{attribute 'GeneratedUsingTerminal: EK1100-0000-0018'}
{attribute addProperty BoxType "EK1100-0000-0018"}
{attribute addProperty Id "Beckhoff_EL4xxxEK1122Beckhoff_EL4xxxEK1122_243FD9A62A_0001_EL4001_0000_0016EL4001_2FC30C535A_0002_EL4001_0000_0017EL4001_2FC30C535A_0003_EL4001_0000_0018EL4001_2FC30C535A_0004_EL4001_0000_0019EL4001_2FC30C535A_0005_EL4001_0000_0020EL4001_2FC30C535A_0006_EL4002_0000_0016EL4002_CAB4C8F57A_0007_EL4002_0000_0017EL4002_CAB4C8F57A_0008_EL4002_0000_0018EL4002_D295D1387A_0009_EL4002_0000_0019EL4002_CAB4C8F57A_0010_EL4002_0000_0020EL4002_CAB4C8F57A_0011_EL4004_0000_0016EL4004_EB925BA911A_0012_EL4004_0000_0017EL4004_EB925BA911A_0013_EL4004_0000_0018EL4004_57A43C6411A_0014_EL4004_0000_0019EL4004_EB925BA911A_0015_EL4004_0000_0020EL4004_EB925BA911A_0016_EL4008_0000_0016EL4008_9E80CF7619A_0017_EL4008_0000_0017EL4008_9E80CF7619A_0018_EL4008_0000_0018EL4008_8B2492A319A_0019_EL4008_0000_0019EL4008_9E80CF7619A_0020_EL4008_0000_0020EL4008_9E80CF7619A_0021_EL4011_0000_0016EL4011_2FC30C535A_0022_EL4011_0000_0017EL4011_2FC30C535A_0023_EL4011_0000_0018EL4011_2FC30C535A_0024_EL4011_0000_0019EL4011_2FC30C535A_0025_EL4011_0000_0020EL4011_2FC30C535A_0026_EL4012_0000_0016EL4012_CAB4C8F57A_0027_EL4012_0000_0017EL4012_CAB4C8F57A_0028_EL4012_0000_0018EL4012_D295D1387A_0029_EL4012_0000_0019EL4012_CAB4C8F57A_0030_EL4012_0000_0020EL4012_CAB4C8F57A_0031_EL4014_0000_0016EL4014_EB925BA911A_0032_EL4014_0000_0017EL4014_EB925BA911A_0033_EL4014_0000_0018EL4014_57A43C6411A_0034_EL4014_0000_0019EL4014_EB925BA911A_0035_EL4014_0000_0020EL4014_EB925BA911A_0036_EL4018_0000_0016EL4018_9E80CF7619A_0037_EL4018_0000_0017EL4018_9E80CF7619A_0038_EL4018_0000_0018EL4018_8B2492A319A_0039_EL4018_0000_0019EL4018_9E80CF7619A_0040_EL4018_0000_0020EL4018_9E80CF7619A_0041_EL4021_0000_0016EL4021_2FC30C535A_0042_EL4021_0000_0017EL4021_2FC30C535A_0043_EL4021_0000_0018EL4021_2FC30C535A_0044_EL4021_0000_0019EL4021_2FC30C535A_0045_EL4021_0000_0020EL4021_2FC30C535A_0046_EL4021_0000_0021EL4021_2FC30C535A_0047_EL4022_0000_0016EL4022_CAB4C8F57A_0048_EL4022_0000_0017EL4022_CAB4C8F57A_0049_EL4022_0000_0018EL4022_D295D1387A_0050_EL4022_0000_0019EL4022_CAB4C8F57A_0051_EL4022_0000_0020EL4022_CAB4C8F57A_0052_EL4022_0000_0021EL4022_CAB4C8F57A_0053_EL4024_0000_0016EL4024_EB925BA911A_0054_EL4024_0000_0017EL4024_EB925BA911A_0055_EL4024_0000_0018EL4024_57A43C6411A_0056_EL4024_0000_0019EL4024_EB925BA911A_0057_EL4024_0000_0020EL4024_EB925BA911A_0058_EL4024_0000_0021EL4024_EB925BA911A_0059_EL4028_0000_0016EL4028_9E80CF7619A_0060_EL4028_0000_0017EL4028_9E80CF7619A_0061_EL4028_0000_0018EL4028_8B2492A319A_0062_EL4028_0000_0019EL4028_9E80CF7619A_0063_EL4028_0000_0020EL4028_9E80CF7619A_0064_EL4028_0000_0021EL4028_9E80CF7619A_0065_EL4031_0000_0016EL4031_2FC30C535A_0066_EL4031_0000_0017EL4031_2FC30C535A_0067_EL4031_0000_0018EL4031_2FC30C535A_0068_EL4031_0000_0019EL4031_2FC30C535A_0069_EL4031_0000_0020EL4031_2FC30C535A_0070_EL4032_0000_0016EL4032_CAB4C8F57A_0071_EL4032_0000_0017EL4032_CAB4C8F57A_0072_EL4032_0000_0018EL4032_D295D1387A_0073_EL4032_0000_0019EL4032_CAB4C8F57A_0074_EL4032_0000_0020EL4032_CAB4C8F57A_0075_EL4034_0000_0016EL4034_EB925BA911A_0076_EL4034_0000_0017EL4034_EB925BA911A_0077_EL4034_0000_0018EL4034_57A43C6411A_0078_EL4034_0000_0019EL4034_EB925BA911A_0079_EL4034_0000_0020EL4034_EB925BA911A_0080_EL4038_0000_0016EL4038_9E80CF7619A_0081_EL4038_0000_0017EL4038_9E80CF7619A_0082_EL4038_0000_0018EL4038_8B2492A319A_0083_EL4038_0000_0019EL4038_9E80CF7619A_0084_EL4038_0000_0020EL4038_9E80CF7619A_0085_EL4102_0000_0000EL4102_DDDE0D3B7A_0086_EL4102_0000_1016EL4102_DDDE0D3B7A_0087_EL4102_0000_1017EL4102_DDDE0D3B7A_0088_EL4102_0000_1018EL4102_DDDE0D3B7A_0089_EL4102_0000_1019EL4102_DDDE0D3B7A_0090_EL4102_0000_1020EL4102_DDDE0D3B7A_0091_EL4104_0000_1016EL4104_57A43C6411A_0092_EL4104_0000_1017EL4104_57A43C6411A_0093_EL4104_0000_1018EL4104_57A43C6411A_0094_EL4104_0000_1019EL4104_57A43C6411A_0095_EL4104_0000_1020EL4104_57A43C6411A_0096_EL4112_0000_0000EL4112_DDDE0D3B7A_0097_EL4112_0000_1016EL4112_DDDE0D3B7A_0098_EL4112_0000_1017EL4112_DDDE0D3B7A_0099_EL4112_0000_1018EL4112_DDDE0D3B7A_0100_EL4112_0000_1019EL4112_DDDE0D3B7A_0101_EL4112_0000_1020EL4112_DDDE0D3B7A_0102_EL4112_0010_0000EL4112_DDDE0D3B7A_0103_EL4112_0010_1016EL4112_DDDE0D3B7A_0104_EL4112_0010_1017EL4112_DDDE0D3B7A_0105_EL4112_0010_1018EL4112_DDDE0D3B7A_0106_EL4112_0010_1019EL4112_DDDE0D3B7A_0107_EL4112_0010_1020EL4112_DDDE0D3B7A_0108_EL4114_0000_1016EL4114_57A43C6411A_0109_EL4114_0000_1017EL4114_57A43C6411A_0110_EL4114_0000_1018EL4114_57A43C6411A_0111_EL4114_0000_1019EL4114_57A43C6411A_0112_EL4114_0000_1020EL4114_57A43C6411A_0113_EL4122_0000_0000EL4122_DDDE0D3B7A_0114_EL4122_0000_1016EL4122_DDDE0D3B7A_0115_EL4122_0000_1017EL4122_DDDE0D3B7A_0116_EL4122_0000_1018EL4122_DDDE0D3B7A_0117_EL4122_0000_1019EL4122_DDDE0D3B7A_0118_EL4122_0000_1020EL4122_DDDE0D3B7A_0119_EL4124_0000_1016EL4124_57A43C6411A_0120_EL4124_0000_1017EL4124_57A43C6411A_0121_EL4124_0000_1018EL4124_57A43C6411A_0122_EL4124_0000_1019EL4124_57A43C6411A_0123_EL4124_0000_1020EL4124_57A43C6411A_0124_EL4132_0000_0000EL4132_DDDE0D3B7A_0125_EL4132_0000_1016EL4132_DDDE0D3B7A_0126_EL4132_0000_1017EL4132_DDDE0D3B7A_0127_EL4132_0000_1018EL4132_DDDE0D3B7A_0128_EL4132_0000_1019EL4132_DDDE0D3B7A_0129_EL4132_0000_1020EL4132_DDDE0D3B7A_0130_EL4134_0000_1016EL4134_57A43C6411A_0131_EL4134_0000_1017EL4134_57A43C6411A_0132_EL4134_0000_1018EL4134_57A43C6411A_0133_EL4134_0000_1019EL4134_57A43C6411A_0134_EL4134_0000_1020EL4134_57A43C6411A_0135_EL4134_0030_1020EL4134_57A43C6411"}
{attribute addProperty CRC "2306607182"}
{attribute addProperty Size "1325"}
TYPE Beckhoff_EL4xxx_897C084E EXTENDS EK1100_1FC0878B :
STRUCT
	{attribute addProperty Name "Beckhoff_EL4xxxEK1122"}
	{attribute addProperty PreviousPort "Beckhoff EL4xxx : B"}
	Beckhoff_EL4xxxEK1122 : Beckhoff_EL4xxxEK1122_243FD9A6;
	{attribute addProperty Name "A_0001_EL4001_0000_0016"}
	{attribute addProperty PreviousPort "Beckhoff EL4xxxEK1122 : C"}
	A_0001_EL4001_0000_0016 : EL4001_2FC30C53;
	{attribute addProperty Name "A_0002_EL4001_0000_0017"}
	{attribute addProperty PreviousPort "A_0001(EL4001-0000-0016) : B"}
	A_0002_EL4001_0000_0017 : EL4001_2FC30C53;
	{attribute addProperty Name "A_0003_EL4001_0000_0018"}
	{attribute addProperty PreviousPort "A_0002(EL4001-0000-0017) : B"}
	A_0003_EL4001_0000_0018 : EL4001_2FC30C53;
	{attribute addProperty Name "A_0004_EL4001_0000_0019"}
	{attribute addProperty PreviousPort "A_0003(EL4001-0000-0018) : B"}
	A_0004_EL4001_0000_0019 : EL4001_2FC30C53;
	{attribute addProperty Name "A_0005_EL4001_0000_0020"}
	{attribute addProperty PreviousPort "A_0004(EL4001-0000-0019) : B"}
	A_0005_EL4001_0000_0020 : EL4001_2FC30C53;
	{attribute addProperty Name "A_0006_EL4002_0000_0016"}
	{attribute addProperty PreviousPort "A_0005(EL4001-0000-0020) : B"}
	A_0006_EL4002_0000_0016 : EL4002_CAB4C8F5;
	{attribute addProperty Name "A_0007_EL4002_0000_0017"}
	{attribute addProperty PreviousPort "A_0006(EL4002-0000-0016) : B"}
	A_0007_EL4002_0000_0017 : EL4002_CAB4C8F5;
	{attribute addProperty Name "A_0008_EL4002_0000_0018"}
	{attribute addProperty PreviousPort "A_0007(EL4002-0000-0017) : B"}
	A_0008_EL4002_0000_0018 : EL4002_D295D138;
	{attribute addProperty Name "A_0009_EL4002_0000_0019"}
	{attribute addProperty PreviousPort "A_0008(EL4002-0000-0018) : B"}
	A_0009_EL4002_0000_0019 : EL4002_CAB4C8F5;
	{attribute addProperty Name "A_0010_EL4002_0000_0020"}
	{attribute addProperty PreviousPort "A_0009(EL4002-0000-0019) : B"}
	A_0010_EL4002_0000_0020 : EL4002_CAB4C8F5;
	{attribute addProperty Name "A_0011_EL4004_0000_0016"}
	{attribute addProperty PreviousPort "A_0010(EL4002-0000-0020) : B"}
	A_0011_EL4004_0000_0016 : EL4004_EB925BA9;
	{attribute addProperty Name "A_0012_EL4004_0000_0017"}
	{attribute addProperty PreviousPort "A_0011(EL4004-0000-0016) : B"}
	A_0012_EL4004_0000_0017 : EL4004_EB925BA9;
	{attribute addProperty Name "A_0013_EL4004_0000_0018"}
	{attribute addProperty PreviousPort "A_0012(EL4004-0000-0017) : B"}
	A_0013_EL4004_0000_0018 : EL4004_57A43C64;
	{attribute addProperty Name "A_0014_EL4004_0000_0019"}
	{attribute addProperty PreviousPort "A_0013(EL4004-0000-0018) : B"}
	A_0014_EL4004_0000_0019 : EL4004_EB925BA9;
	{attribute addProperty Name "A_0015_EL4004_0000_0020"}
	{attribute addProperty PreviousPort "A_0014(EL4004-0000-0019) : B"}
	A_0015_EL4004_0000_0020 : EL4004_EB925BA9;
	{attribute addProperty Name "A_0016_EL4008_0000_0016"}
	{attribute addProperty PreviousPort "A_0015(EL4004-0000-0020) : B"}
	A_0016_EL4008_0000_0016 : EL4008_9E80CF76;
	{attribute addProperty Name "A_0017_EL4008_0000_0017"}
	{attribute addProperty PreviousPort "A_0016(EL4008-0000-0016) : B"}
	A_0017_EL4008_0000_0017 : EL4008_9E80CF76;
	{attribute addProperty Name "A_0018_EL4008_0000_0018"}
	{attribute addProperty PreviousPort "A_0017(EL4008-0000-0017) : B"}
	A_0018_EL4008_0000_0018 : EL4008_8B2492A3;
	{attribute addProperty Name "A_0019_EL4008_0000_0019"}
	{attribute addProperty PreviousPort "A_0018(EL4008-0000-0018) : B"}
	A_0019_EL4008_0000_0019 : EL4008_9E80CF76;
	{attribute addProperty Name "A_0020_EL4008_0000_0020"}
	{attribute addProperty PreviousPort "A_0019(EL4008-0000-0019) : B"}
	A_0020_EL4008_0000_0020 : EL4008_9E80CF76;
	{attribute addProperty Name "A_0021_EL4011_0000_0016"}
	{attribute addProperty PreviousPort "A_0020(EL4008-0000-0020) : B"}
	A_0021_EL4011_0000_0016 : EL4011_2FC30C53;
	{attribute addProperty Name "A_0022_EL4011_0000_0017"}
	{attribute addProperty PreviousPort "A_0021(EL4011-0000-0016) : B"}
	A_0022_EL4011_0000_0017 : EL4011_2FC30C53;
	{attribute addProperty Name "A_0023_EL4011_0000_0018"}
	{attribute addProperty PreviousPort "A_0022(EL4011-0000-0017) : B"}
	A_0023_EL4011_0000_0018 : EL4011_2FC30C53;
	{attribute addProperty Name "A_0024_EL4011_0000_0019"}
	{attribute addProperty PreviousPort "A_0023(EL4011-0000-0018) : B"}
	A_0024_EL4011_0000_0019 : EL4011_2FC30C53;
	{attribute addProperty Name "A_0025_EL4011_0000_0020"}
	{attribute addProperty PreviousPort "A_0024(EL4011-0000-0019) : B"}
	A_0025_EL4011_0000_0020 : EL4011_2FC30C53;
	{attribute addProperty Name "A_0026_EL4012_0000_0016"}
	{attribute addProperty PreviousPort "A_0025(EL4011-0000-0020) : B"}
	A_0026_EL4012_0000_0016 : EL4012_CAB4C8F5;
	{attribute addProperty Name "A_0027_EL4012_0000_0017"}
	{attribute addProperty PreviousPort "A_0026(EL4012-0000-0016) : B"}
	A_0027_EL4012_0000_0017 : EL4012_CAB4C8F5;
	{attribute addProperty Name "A_0028_EL4012_0000_0018"}
	{attribute addProperty PreviousPort "A_0027(EL4012-0000-0017) : B"}
	A_0028_EL4012_0000_0018 : EL4012_D295D138;
	{attribute addProperty Name "A_0029_EL4012_0000_0019"}
	{attribute addProperty PreviousPort "A_0028(EL4012-0000-0018) : B"}
	A_0029_EL4012_0000_0019 : EL4012_CAB4C8F5;
	{attribute addProperty Name "A_0030_EL4012_0000_0020"}
	{attribute addProperty PreviousPort "A_0029(EL4012-0000-0019) : B"}
	A_0030_EL4012_0000_0020 : EL4012_CAB4C8F5;
	{attribute addProperty Name "A_0031_EL4014_0000_0016"}
	{attribute addProperty PreviousPort "A_0030(EL4012-0000-0020) : B"}
	A_0031_EL4014_0000_0016 : EL4014_EB925BA9;
	{attribute addProperty Name "A_0032_EL4014_0000_0017"}
	{attribute addProperty PreviousPort "A_0031(EL4014-0000-0016) : B"}
	A_0032_EL4014_0000_0017 : EL4014_EB925BA9;
	{attribute addProperty Name "A_0033_EL4014_0000_0018"}
	{attribute addProperty PreviousPort "A_0032(EL4014-0000-0017) : B"}
	A_0033_EL4014_0000_0018 : EL4014_57A43C64;
	{attribute addProperty Name "A_0034_EL4014_0000_0019"}
	{attribute addProperty PreviousPort "A_0033(EL4014-0000-0018) : B"}
	A_0034_EL4014_0000_0019 : EL4014_EB925BA9;
	{attribute addProperty Name "A_0035_EL4014_0000_0020"}
	{attribute addProperty PreviousPort "A_0034(EL4014-0000-0019) : B"}
	A_0035_EL4014_0000_0020 : EL4014_EB925BA9;
	{attribute addProperty Name "A_0036_EL4018_0000_0016"}
	{attribute addProperty PreviousPort "A_0035(EL4014-0000-0020) : B"}
	A_0036_EL4018_0000_0016 : EL4018_9E80CF76;
	{attribute addProperty Name "A_0037_EL4018_0000_0017"}
	{attribute addProperty PreviousPort "A_0036(EL4018-0000-0016) : B"}
	A_0037_EL4018_0000_0017 : EL4018_9E80CF76;
	{attribute addProperty Name "A_0038_EL4018_0000_0018"}
	{attribute addProperty PreviousPort "A_0037(EL4018-0000-0017) : B"}
	A_0038_EL4018_0000_0018 : EL4018_8B2492A3;
	{attribute addProperty Name "A_0039_EL4018_0000_0019"}
	{attribute addProperty PreviousPort "A_0038(EL4018-0000-0018) : B"}
	A_0039_EL4018_0000_0019 : EL4018_9E80CF76;
	{attribute addProperty Name "A_0040_EL4018_0000_0020"}
	{attribute addProperty PreviousPort "A_0039(EL4018-0000-0019) : B"}
	A_0040_EL4018_0000_0020 : EL4018_9E80CF76;
	{attribute addProperty Name "A_0041_EL4021_0000_0016"}
	{attribute addProperty PreviousPort "A_0040(EL4018-0000-0020) : B"}
	A_0041_EL4021_0000_0016 : EL4021_2FC30C53;
	{attribute addProperty Name "A_0042_EL4021_0000_0017"}
	{attribute addProperty PreviousPort "A_0041(EL4021-0000-0016) : B"}
	A_0042_EL4021_0000_0017 : EL4021_2FC30C53;
	{attribute addProperty Name "A_0043_EL4021_0000_0018"}
	{attribute addProperty PreviousPort "A_0042(EL4021-0000-0017) : B"}
	A_0043_EL4021_0000_0018 : EL4021_2FC30C53;
	{attribute addProperty Name "A_0044_EL4021_0000_0019"}
	{attribute addProperty PreviousPort "A_0043(EL4021-0000-0018) : B"}
	A_0044_EL4021_0000_0019 : EL4021_2FC30C53;
	{attribute addProperty Name "A_0045_EL4021_0000_0020"}
	{attribute addProperty PreviousPort "A_0044(EL4021-0000-0019) : B"}
	A_0045_EL4021_0000_0020 : EL4021_2FC30C53;
	{attribute addProperty Name "A_0046_EL4021_0000_0021"}
	{attribute addProperty PreviousPort "A_0045(EL4021-0000-0020) : B"}
	A_0046_EL4021_0000_0021 : EL4021_2FC30C53;
	{attribute addProperty Name "A_0047_EL4022_0000_0016"}
	{attribute addProperty PreviousPort "A_0046(EL4021-0000-0021) : B"}
	A_0047_EL4022_0000_0016 : EL4022_CAB4C8F5;
	{attribute addProperty Name "A_0048_EL4022_0000_0017"}
	{attribute addProperty PreviousPort "A_0047(EL4022-0000-0016) : B"}
	A_0048_EL4022_0000_0017 : EL4022_CAB4C8F5;
	{attribute addProperty Name "A_0049_EL4022_0000_0018"}
	{attribute addProperty PreviousPort "A_0048(EL4022-0000-0017) : B"}
	A_0049_EL4022_0000_0018 : EL4022_D295D138;
	{attribute addProperty Name "A_0050_EL4022_0000_0019"}
	{attribute addProperty PreviousPort "A_0049(EL4022-0000-0018) : B"}
	A_0050_EL4022_0000_0019 : EL4022_CAB4C8F5;
	{attribute addProperty Name "A_0051_EL4022_0000_0020"}
	{attribute addProperty PreviousPort "A_0050(EL4022-0000-0019) : B"}
	A_0051_EL4022_0000_0020 : EL4022_CAB4C8F5;
	{attribute addProperty Name "A_0052_EL4022_0000_0021"}
	{attribute addProperty PreviousPort "A_0051(EL4022-0000-0020) : B"}
	A_0052_EL4022_0000_0021 : EL4022_CAB4C8F5;
	{attribute addProperty Name "A_0053_EL4024_0000_0016"}
	{attribute addProperty PreviousPort "A_0052(EL4022-0000-0021) : B"}
	A_0053_EL4024_0000_0016 : EL4024_EB925BA9;
	{attribute addProperty Name "A_0054_EL4024_0000_0017"}
	{attribute addProperty PreviousPort "A_0053(EL4024-0000-0016) : B"}
	A_0054_EL4024_0000_0017 : EL4024_EB925BA9;
	{attribute addProperty Name "A_0055_EL4024_0000_0018"}
	{attribute addProperty PreviousPort "A_0054(EL4024-0000-0017) : B"}
	A_0055_EL4024_0000_0018 : EL4024_57A43C64;
	{attribute addProperty Name "A_0056_EL4024_0000_0019"}
	{attribute addProperty PreviousPort "A_0055(EL4024-0000-0018) : B"}
	A_0056_EL4024_0000_0019 : EL4024_EB925BA9;
	{attribute addProperty Name "A_0057_EL4024_0000_0020"}
	{attribute addProperty PreviousPort "A_0056(EL4024-0000-0019) : B"}
	A_0057_EL4024_0000_0020 : EL4024_EB925BA9;
	{attribute addProperty Name "A_0058_EL4024_0000_0021"}
	{attribute addProperty PreviousPort "A_0057(EL4024-0000-0020) : B"}
	A_0058_EL4024_0000_0021 : EL4024_EB925BA9;
	{attribute addProperty Name "A_0059_EL4028_0000_0016"}
	{attribute addProperty PreviousPort "A_0058(EL4024-0000-0021) : B"}
	A_0059_EL4028_0000_0016 : EL4028_9E80CF76;
	{attribute addProperty Name "A_0060_EL4028_0000_0017"}
	{attribute addProperty PreviousPort "A_0059(EL4028-0000-0016) : B"}
	A_0060_EL4028_0000_0017 : EL4028_9E80CF76;
	{attribute addProperty Name "A_0061_EL4028_0000_0018"}
	{attribute addProperty PreviousPort "A_0060(EL4028-0000-0017) : B"}
	A_0061_EL4028_0000_0018 : EL4028_8B2492A3;
	{attribute addProperty Name "A_0062_EL4028_0000_0019"}
	{attribute addProperty PreviousPort "A_0061(EL4028-0000-0018) : B"}
	A_0062_EL4028_0000_0019 : EL4028_9E80CF76;
	{attribute addProperty Name "A_0063_EL4028_0000_0020"}
	{attribute addProperty PreviousPort "A_0062(EL4028-0000-0019) : B"}
	A_0063_EL4028_0000_0020 : EL4028_9E80CF76;
	{attribute addProperty Name "A_0064_EL4028_0000_0021"}
	{attribute addProperty PreviousPort "A_0063(EL4028-0000-0020) : B"}
	A_0064_EL4028_0000_0021 : EL4028_9E80CF76;
	{attribute addProperty Name "A_0065_EL4031_0000_0016"}
	{attribute addProperty PreviousPort "A_0064(EL4028-0000-0021) : B"}
	A_0065_EL4031_0000_0016 : EL4031_2FC30C53;
	{attribute addProperty Name "A_0066_EL4031_0000_0017"}
	{attribute addProperty PreviousPort "A_0065(EL4031-0000-0016) : B"}
	A_0066_EL4031_0000_0017 : EL4031_2FC30C53;
	{attribute addProperty Name "A_0067_EL4031_0000_0018"}
	{attribute addProperty PreviousPort "A_0066(EL4031-0000-0017) : B"}
	A_0067_EL4031_0000_0018 : EL4031_2FC30C53;
	{attribute addProperty Name "A_0068_EL4031_0000_0019"}
	{attribute addProperty PreviousPort "A_0067(EL4031-0000-0018) : B"}
	A_0068_EL4031_0000_0019 : EL4031_2FC30C53;
	{attribute addProperty Name "A_0069_EL4031_0000_0020"}
	{attribute addProperty PreviousPort "A_0068(EL4031-0000-0019) : B"}
	A_0069_EL4031_0000_0020 : EL4031_2FC30C53;
	{attribute addProperty Name "A_0070_EL4032_0000_0016"}
	{attribute addProperty PreviousPort "A_0069(EL4031-0000-0020) : B"}
	A_0070_EL4032_0000_0016 : EL4032_CAB4C8F5;
	{attribute addProperty Name "A_0071_EL4032_0000_0017"}
	{attribute addProperty PreviousPort "A_0070(EL4032-0000-0016) : B"}
	A_0071_EL4032_0000_0017 : EL4032_CAB4C8F5;
	{attribute addProperty Name "A_0072_EL4032_0000_0018"}
	{attribute addProperty PreviousPort "A_0071(EL4032-0000-0017) : B"}
	A_0072_EL4032_0000_0018 : EL4032_D295D138;
	{attribute addProperty Name "A_0073_EL4032_0000_0019"}
	{attribute addProperty PreviousPort "A_0072(EL4032-0000-0018) : B"}
	A_0073_EL4032_0000_0019 : EL4032_CAB4C8F5;
	{attribute addProperty Name "A_0074_EL4032_0000_0020"}
	{attribute addProperty PreviousPort "A_0073(EL4032-0000-0019) : B"}
	A_0074_EL4032_0000_0020 : EL4032_CAB4C8F5;
	{attribute addProperty Name "A_0075_EL4034_0000_0016"}
	{attribute addProperty PreviousPort "A_0074(EL4032-0000-0020) : B"}
	A_0075_EL4034_0000_0016 : EL4034_EB925BA9;
	{attribute addProperty Name "A_0076_EL4034_0000_0017"}
	{attribute addProperty PreviousPort "A_0075(EL4034-0000-0016) : B"}
	A_0076_EL4034_0000_0017 : EL4034_EB925BA9;
	{attribute addProperty Name "A_0077_EL4034_0000_0018"}
	{attribute addProperty PreviousPort "A_0076(EL4034-0000-0017) : B"}
	A_0077_EL4034_0000_0018 : EL4034_57A43C64;
	{attribute addProperty Name "A_0078_EL4034_0000_0019"}
	{attribute addProperty PreviousPort "A_0077(EL4034-0000-0018) : B"}
	A_0078_EL4034_0000_0019 : EL4034_EB925BA9;
	{attribute addProperty Name "A_0079_EL4034_0000_0020"}
	{attribute addProperty PreviousPort "A_0078(EL4034-0000-0019) : B"}
	A_0079_EL4034_0000_0020 : EL4034_EB925BA9;
	{attribute addProperty Name "A_0080_EL4038_0000_0016"}
	{attribute addProperty PreviousPort "A_0079(EL4034-0000-0020) : B"}
	A_0080_EL4038_0000_0016 : EL4038_9E80CF76;
	{attribute addProperty Name "A_0081_EL4038_0000_0017"}
	{attribute addProperty PreviousPort "A_0080(EL4038-0000-0016) : B"}
	A_0081_EL4038_0000_0017 : EL4038_9E80CF76;
	{attribute addProperty Name "A_0082_EL4038_0000_0018"}
	{attribute addProperty PreviousPort "A_0081(EL4038-0000-0017) : B"}
	A_0082_EL4038_0000_0018 : EL4038_8B2492A3;
	{attribute addProperty Name "A_0083_EL4038_0000_0019"}
	{attribute addProperty PreviousPort "A_0082(EL4038-0000-0018) : B"}
	A_0083_EL4038_0000_0019 : EL4038_9E80CF76;
	{attribute addProperty Name "A_0084_EL4038_0000_0020"}
	{attribute addProperty PreviousPort "A_0083(EL4038-0000-0019) : B"}
	A_0084_EL4038_0000_0020 : EL4038_9E80CF76;
	{attribute addProperty Name "A_0085_EL4102_0000_0000"}
	{attribute addProperty PreviousPort "A_0084(EL4038-0000-0020) : B"}
	A_0085_EL4102_0000_0000 : EL4102_DDDE0D3B;
	{attribute addProperty Name "A_0086_EL4102_0000_1016"}
	{attribute addProperty PreviousPort "A_0085(EL4102-0000-0000) : B"}
	A_0086_EL4102_0000_1016 : EL4102_DDDE0D3B;
	{attribute addProperty Name "A_0087_EL4102_0000_1017"}
	{attribute addProperty PreviousPort "A_0086(EL4102-0000-1016) : B"}
	A_0087_EL4102_0000_1017 : EL4102_DDDE0D3B;
	{attribute addProperty Name "A_0088_EL4102_0000_1018"}
	{attribute addProperty PreviousPort "A_0087(EL4102-0000-1017) : B"}
	A_0088_EL4102_0000_1018 : EL4102_DDDE0D3B;
	{attribute addProperty Name "A_0089_EL4102_0000_1019"}
	{attribute addProperty PreviousPort "A_0088(EL4102-0000-1018) : B"}
	A_0089_EL4102_0000_1019 : EL4102_DDDE0D3B;
	{attribute addProperty Name "A_0090_EL4102_0000_1020"}
	{attribute addProperty PreviousPort "A_0089(EL4102-0000-1019) : B"}
	A_0090_EL4102_0000_1020 : EL4102_DDDE0D3B;
	{attribute addProperty Name "A_0091_EL4104_0000_1016"}
	{attribute addProperty PreviousPort "A_0090(EL4102-0000-1020) : B"}
	A_0091_EL4104_0000_1016 : EL4104_57A43C64;
	{attribute addProperty Name "A_0092_EL4104_0000_1017"}
	{attribute addProperty PreviousPort "A_0091(EL4104-0000-1016) : B"}
	A_0092_EL4104_0000_1017 : EL4104_57A43C64;
	{attribute addProperty Name "A_0093_EL4104_0000_1018"}
	{attribute addProperty PreviousPort "A_0092(EL4104-0000-1017) : B"}
	A_0093_EL4104_0000_1018 : EL4104_57A43C64;
	{attribute addProperty Name "A_0094_EL4104_0000_1019"}
	{attribute addProperty PreviousPort "A_0093(EL4104-0000-1018) : B"}
	A_0094_EL4104_0000_1019 : EL4104_57A43C64;
	{attribute addProperty Name "A_0095_EL4104_0000_1020"}
	{attribute addProperty PreviousPort "A_0094(EL4104-0000-1019) : B"}
	A_0095_EL4104_0000_1020 : EL4104_57A43C64;
	{attribute addProperty Name "A_0096_EL4112_0000_0000"}
	{attribute addProperty PreviousPort "A_0095(EL4104-0000-1020) : B"}
	A_0096_EL4112_0000_0000 : EL4112_DDDE0D3B;
	{attribute addProperty Name "A_0097_EL4112_0000_1016"}
	{attribute addProperty PreviousPort "A_0096(EL4112-0000-0000) : B"}
	A_0097_EL4112_0000_1016 : EL4112_DDDE0D3B;
	{attribute addProperty Name "A_0098_EL4112_0000_1017"}
	{attribute addProperty PreviousPort "A_0097(EL4112-0000-1016) : B"}
	A_0098_EL4112_0000_1017 : EL4112_DDDE0D3B;
	{attribute addProperty Name "A_0099_EL4112_0000_1018"}
	{attribute addProperty PreviousPort "A_0098(EL4112-0000-1017) : B"}
	A_0099_EL4112_0000_1018 : EL4112_DDDE0D3B;
	{attribute addProperty Name "A_0100_EL4112_0000_1019"}
	{attribute addProperty PreviousPort "A_0099(EL4112-0000-1018) : B"}
	A_0100_EL4112_0000_1019 : EL4112_DDDE0D3B;
	{attribute addProperty Name "A_0101_EL4112_0000_1020"}
	{attribute addProperty PreviousPort "A_0100(EL4112-0000-1019) : B"}
	A_0101_EL4112_0000_1020 : EL4112_DDDE0D3B;
	{attribute addProperty Name "A_0102_EL4112_0010_0000"}
	{attribute addProperty PreviousPort "A_0101(EL4112-0000-1020) : B"}
	A_0102_EL4112_0010_0000 : EL4112_DDDE0D3B;
	{attribute addProperty Name "A_0103_EL4112_0010_1016"}
	{attribute addProperty PreviousPort "A_0102(EL4112-0010-0000) : B"}
	A_0103_EL4112_0010_1016 : EL4112_DDDE0D3B;
	{attribute addProperty Name "A_0104_EL4112_0010_1017"}
	{attribute addProperty PreviousPort "A_0103(EL4112-0010-1016) : B"}
	A_0104_EL4112_0010_1017 : EL4112_DDDE0D3B;
	{attribute addProperty Name "A_0105_EL4112_0010_1018"}
	{attribute addProperty PreviousPort "A_0104(EL4112-0010-1017) : B"}
	A_0105_EL4112_0010_1018 : EL4112_DDDE0D3B;
	{attribute addProperty Name "A_0106_EL4112_0010_1019"}
	{attribute addProperty PreviousPort "A_0105(EL4112-0010-1018) : B"}
	A_0106_EL4112_0010_1019 : EL4112_DDDE0D3B;
	{attribute addProperty Name "A_0107_EL4112_0010_1020"}
	{attribute addProperty PreviousPort "A_0106(EL4112-0010-1019) : B"}
	A_0107_EL4112_0010_1020 : EL4112_DDDE0D3B;
	{attribute addProperty Name "A_0108_EL4114_0000_1016"}
	{attribute addProperty PreviousPort "A_0107(EL4112-0010-1020) : B"}
	A_0108_EL4114_0000_1016 : EL4114_57A43C64;
	{attribute addProperty Name "A_0109_EL4114_0000_1017"}
	{attribute addProperty PreviousPort "A_0108(EL4114-0000-1016) : B"}
	A_0109_EL4114_0000_1017 : EL4114_57A43C64;
	{attribute addProperty Name "A_0110_EL4114_0000_1018"}
	{attribute addProperty PreviousPort "A_0109(EL4114-0000-1017) : B"}
	A_0110_EL4114_0000_1018 : EL4114_57A43C64;
	{attribute addProperty Name "A_0111_EL4114_0000_1019"}
	{attribute addProperty PreviousPort "A_0110(EL4114-0000-1018) : B"}
	A_0111_EL4114_0000_1019 : EL4114_57A43C64;
	{attribute addProperty Name "A_0112_EL4114_0000_1020"}
	{attribute addProperty PreviousPort "A_0111(EL4114-0000-1019) : B"}
	A_0112_EL4114_0000_1020 : EL4114_57A43C64;
	{attribute addProperty Name "A_0113_EL4122_0000_0000"}
	{attribute addProperty PreviousPort "A_0112(EL4114-0000-1020) : B"}
	A_0113_EL4122_0000_0000 : EL4122_DDDE0D3B;
	{attribute addProperty Name "A_0114_EL4122_0000_1016"}
	{attribute addProperty PreviousPort "A_0113(EL4122-0000-0000) : B"}
	A_0114_EL4122_0000_1016 : EL4122_DDDE0D3B;
	{attribute addProperty Name "A_0115_EL4122_0000_1017"}
	{attribute addProperty PreviousPort "A_0114(EL4122-0000-1016) : B"}
	A_0115_EL4122_0000_1017 : EL4122_DDDE0D3B;
	{attribute addProperty Name "A_0116_EL4122_0000_1018"}
	{attribute addProperty PreviousPort "A_0115(EL4122-0000-1017) : B"}
	A_0116_EL4122_0000_1018 : EL4122_DDDE0D3B;
	{attribute addProperty Name "A_0117_EL4122_0000_1019"}
	{attribute addProperty PreviousPort "A_0116(EL4122-0000-1018) : B"}
	A_0117_EL4122_0000_1019 : EL4122_DDDE0D3B;
	{attribute addProperty Name "A_0118_EL4122_0000_1020"}
	{attribute addProperty PreviousPort "A_0117(EL4122-0000-1019) : B"}
	A_0118_EL4122_0000_1020 : EL4122_DDDE0D3B;
	{attribute addProperty Name "A_0119_EL4124_0000_1016"}
	{attribute addProperty PreviousPort "A_0118(EL4122-0000-1020) : B"}
	A_0119_EL4124_0000_1016 : EL4124_57A43C64;
	{attribute addProperty Name "A_0120_EL4124_0000_1017"}
	{attribute addProperty PreviousPort "A_0119(EL4124-0000-1016) : B"}
	A_0120_EL4124_0000_1017 : EL4124_57A43C64;
	{attribute addProperty Name "A_0121_EL4124_0000_1018"}
	{attribute addProperty PreviousPort "A_0120(EL4124-0000-1017) : B"}
	A_0121_EL4124_0000_1018 : EL4124_57A43C64;
	{attribute addProperty Name "A_0122_EL4124_0000_1019"}
	{attribute addProperty PreviousPort "A_0121(EL4124-0000-1018) : B"}
	A_0122_EL4124_0000_1019 : EL4124_57A43C64;
	{attribute addProperty Name "A_0123_EL4124_0000_1020"}
	{attribute addProperty PreviousPort "A_0122(EL4124-0000-1019) : B"}
	A_0123_EL4124_0000_1020 : EL4124_57A43C64;
	{attribute addProperty Name "A_0124_EL4132_0000_0000"}
	{attribute addProperty PreviousPort "A_0123(EL4124-0000-1020) : B"}
	A_0124_EL4132_0000_0000 : EL4132_DDDE0D3B;
	{attribute addProperty Name "A_0125_EL4132_0000_1016"}
	{attribute addProperty PreviousPort "A_0124(EL4132-0000-0000) : B"}
	A_0125_EL4132_0000_1016 : EL4132_DDDE0D3B;
	{attribute addProperty Name "A_0126_EL4132_0000_1017"}
	{attribute addProperty PreviousPort "A_0125(EL4132-0000-1016) : B"}
	A_0126_EL4132_0000_1017 : EL4132_DDDE0D3B;
	{attribute addProperty Name "A_0127_EL4132_0000_1018"}
	{attribute addProperty PreviousPort "A_0126(EL4132-0000-1017) : B"}
	A_0127_EL4132_0000_1018 : EL4132_DDDE0D3B;
	{attribute addProperty Name "A_0128_EL4132_0000_1019"}
	{attribute addProperty PreviousPort "A_0127(EL4132-0000-1018) : B"}
	A_0128_EL4132_0000_1019 : EL4132_DDDE0D3B;
	{attribute addProperty Name "A_0129_EL4132_0000_1020"}
	{attribute addProperty PreviousPort "A_0128(EL4132-0000-1019) : B"}
	A_0129_EL4132_0000_1020 : EL4132_DDDE0D3B;
	{attribute addProperty Name "A_0130_EL4134_0000_1016"}
	{attribute addProperty PreviousPort "A_0129(EL4132-0000-1020) : B"}
	A_0130_EL4134_0000_1016 : EL4134_57A43C64;
	{attribute addProperty Name "A_0131_EL4134_0000_1017"}
	{attribute addProperty PreviousPort "A_0130(EL4134-0000-1016) : B"}
	A_0131_EL4134_0000_1017 : EL4134_57A43C64;
	{attribute addProperty Name "A_0132_EL4134_0000_1018"}
	{attribute addProperty PreviousPort "A_0131(EL4134-0000-1017) : B"}
	A_0132_EL4134_0000_1018 : EL4134_57A43C64;
	{attribute addProperty Name "A_0133_EL4134_0000_1019"}
	{attribute addProperty PreviousPort "A_0132(EL4134-0000-1018) : B"}
	A_0133_EL4134_0000_1019 : EL4134_57A43C64;
	{attribute addProperty Name "A_0134_EL4134_0000_1020"}
	{attribute addProperty PreviousPort "A_0133(EL4134-0000-1019) : B"}
	A_0134_EL4134_0000_1020 : EL4134_57A43C64;
	{attribute addProperty Name "A_0135_EL4134_0030_1020"}
	{attribute addProperty PreviousPort "A_0134(EL4134-0000-1020) : B"}
	A_0135_EL4134_0030_1020 : EL4134_57A43C64;
END_STRUCT
END_TYPE

(* stored: Version 1.2.0.0, ProductVersion 3.1.4024.9
   DUT Beckhoff_EL4xxx_897C084E: Id {21f41368-8f17-4b20-a6e0-184532867566} *)
